RESOURCE_TYPE VIEW_PANEL (* Container for View elements *)
  (* Standard: 61499-1; Classification: HMI *)
  (* Version 0.2, 2006-10-17, JHC, Holobloc Inc, Corrected package in CompilerInfo. *)
  (* Version 0.1, 2006-02-28, JHC, Holobloc Inc, Removed TRACE. *)
  (* Version 0.0, 2002-04-04, JHC, Rockwell Automation, Derived from PANEL_RESOURCE. *)
  (* Compiler header: package fb.rt.mva; *)
  (* Compiler Java Sun JDK 1.6.0 *)
  VAR_INPUT
    BKGD : COLOR := COLOR#white; (* Background color *)
    DIA : UINT := 25; (* Characteristic dimension,Overrides component DIAs *)
    SIZE : ARRAY [0..1] OF UINT := [2,2]; (* [width,height]in DIA units *)
    VERTICAL : BOOL; (* 1=Column-first,0=Row-first *)
  END_VAR
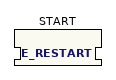
  FBS
    START : E_RESTART;
  END_FBS
END_RESOURCE_TYPE
